{attribute 'qualified_only'}
{attribute 'strict'}
TYPE E_SampleSlotStates :
(
    EMPTY,
    FULL,
    DISABLED
);
END_TYPE

(* stored: Version 1.1.0.1
   DUT E_SampleSlotStates: Id {57679c10-1d31-446b-ab2d-82c03a214142} *)
